(* PLC project , Beckhoff Automation GmbH TwinCAT PLC Control 3.5.13.21 *)
(* stored: creationDateTime 2025-04-03T10:43:18.9008552 *)

FUNCTION_BLOCK FB_DataLogger
VAR_INPUT
    netId       : T_AmsNetId;        // TwinCAT network ID (e.g., '')
    sFileName   : T_MaxString;       // File path and name (e.g., 'C:\Logs\data.bin')
    bOpen       : BOOL;              // Rising edge to trigger file open
    bWrite      : BOOL;              // Rising edge to trigger data write
    bClose      : BOOL;              // Rising edge to trigger file close
    t           : LREAL;             // Timestamp or simulation time
    act_pos     : LREAL;             // Actual position to log
    act_vel     : LREAL;             // Actual velocity to log
    act_torque  : LREAL;             // Actual torque to log
END_VAR
VAR_OUTPUT
    bDone       : BOOL;              // Set TRUE when file is successfully closed
    bBusy       : BOOL;              // Indicates if file operation is in progress
    bError      : BOOL;              // Set TRUE on any error
    nErrorId    : UDINT;             // TwinCAT file function error code
    hFile       : UINT;              // File handle (used for writing/closing)
END_VAR
VAR
    dataBuffer     : ARRAY[1..4] OF LREAL;  // Buffer for logging data
    nBytesToWrite  : UDINT;                 // Number of bytes to write
    fbFileOpen     : FB_FileOpen;           // File open function block
    fbFileWrite    : FB_FileWrite;          // File write function block
    fbFileClose    : FB_FileClose;          // File close function block
    bFileOpen      : BOOL := TRUE;          // Internal flag for open execution control
END_VAR

VAR_TEMP
	
END_VAR

            (*
------------------------------------------------------------------------------
FB_DataLogger - Binary Data Logger Function Block

DESCRIPTION:
This function block logs a set of numerical values (e.g., timestamp, position,
velocity, torque) into a binary file. It is suitable for real-time signal logging
during experiments, simulations, or runtime testing.

FEATURES:
- Handles file opening, writing, and closing internally
- Binary file format using an LREAL array
- 5-second timeout protection for each file operation
- Outputs useful status flags for diagnostics and visualization
- File handle exposed for integration with other blocks

INPUTS:
- netId      : T_AmsNetId  → Network ID (use '' for local)
- sFileName  : T_MaxString → Full path to the file to open/write
- bOpen      : BOOL        → Trigger to open the file
- bWrite     : BOOL        → Trigger to write a data sample
- bClose     : BOOL        → Trigger to close the file
- t          : LREAL       → Time value to log
- act_pos    : LREAL       → Position value to log
- act_vel    : LREAL       → Velocity value to log
- act_torque : LREAL       → Torque value to log

OUTPUTS:
- bDone      : BOOL    → TRUE when file closed successfully
- bBusy      : BOOL    → TRUE when file close is ongoing
- bError     : BOOL    → TRUE if any file operation fails
- nErrorId   : UDINT   → Error code from TwinCAT file functions
- hFile      : UINT    → File handle currently in use

USAGE:
Call this block cyclically. Use rising edge triggers for bOpen, bWrite, and bClose.
Data is written in binary format using `ARRAY[1..4] OF LREAL`. Suitable for analysis
with external tools or for real-time streaming to memory buffers.

VERSION:
v1.0 - March 2025

AUTHOR:
Manuel Beschi cari.unibs.it

------------------------------------------------------------------------------
*)

// === Step 1: Open File ===
IF bOpen THEN
    // Perform a two-step execution to latch rising edge for file open
    fbFileOpen(
        sPathName := sFileName,
        nMode     := FOPEN_MODEWRITE OR FOPEN_MODEBINARY, // Overwrites if exists
        sNetId    := netId,
        bExecute  := FALSE,
        tTimeout  := T#5S // 5 seconds timeout
    );
    fbFileOpen(
        sPathName := sFileName,
        nMode     := FOPEN_MODEWRITE OR FOPEN_MODEBINARY,
        sNetId    := netId,
        bExecute  := TRUE,
        tTimeout  := T#5S // 5 seconds timeout
    );

    // Check file open result
    IF NOT fbFileOpen.bBusy THEN
        IF NOT fbFileOpen.bError THEN
            hFile := fbFileOpen.hFile;
            bOpen := FALSE; // Reset trigger
        ELSE
            bError := TRUE;
            nErrorId := fbFileOpen.nErrId;
        END_IF
    END_IF
END_IF

// Safety check if open is still busy (extra safe check)
IF fbFileOpen.bBusy THEN
    fbFileOpen(); // Call again to keep evaluating
    IF NOT fbFileOpen.bError THEN
        hFile := fbFileOpen.hFile;
        bOpen := FALSE;
    ELSE
        bError := TRUE;
        nErrorId := fbFileOpen.nErrId;
    END_IF
END_IF

// === Step 2: Write Data ===
IF bWrite AND (NOT fbFileOpen.bBusy) THEN
    // Prepare data buffer with current inputs
    dataBuffer[1] := t;
    dataBuffer[2] := act_pos;
    dataBuffer[3] := act_vel;
    dataBuffer[4] := act_torque;

    nBytesToWrite := SIZEOF(dataBuffer); // Size in bytes

    // Do a two-step write with rising edge simulation
    fbFileWrite(
        sNetId      := netId,
        hFile       := hFile,
        pWriteBuff  := ADR(dataBuffer),
        cbWriteLen  := nBytesToWrite,
        bExecute    := FALSE
    );
    fbFileWrite(
        sNetId      := netId,
        hFile       := hFile,
        pWriteBuff  := ADR(dataBuffer),
        cbWriteLen  := nBytesToWrite,
        bExecute    := TRUE
    );
END_IF

// === Step 3: Close File ===
IF bClose THEN
    fbFileClose.bExecute := FALSE; // Rising edge handling

    // Execute close operation
    fbFileClose(
        hFile     := hFile,
        bExecute  := TRUE,
        tTimeout  := T#5S
    );

    // Output states
    bBusy := fbFileClose.bBusy;
    bError := fbFileClose.bError;
    nErrorId := fbFileClose.nErrId;

    // Check if closed successfully
    IF NOT fbFileClose.bBusy THEN
        IF NOT fbFileClose.bError THEN
            bClose := FALSE;
            bDone := TRUE;
            hFile := 0; // Invalidate handle
        END_IF
    END_IF
ELSE
    bDone := FALSE; // Clear done when not closing
END_IF


          
END_FUNCTION_BLOCK
